TYPE "PL_DigIntlock"
VERSION : 0.1
   STRUCT
      Value { ExternalVisible := 'False'} : Bool;
      BypAct { ExternalVisible := 'False'} : Bool;
      ST { ExternalVisible := 'False'} : Byte := 16#FF;
   END_STRUCT;

END_TYPE

